// LS Electric XG5000 project: 0201 선풍기
// PLC LSPLC

PROGRAM NewProgram (task: 스캔 프로그램)

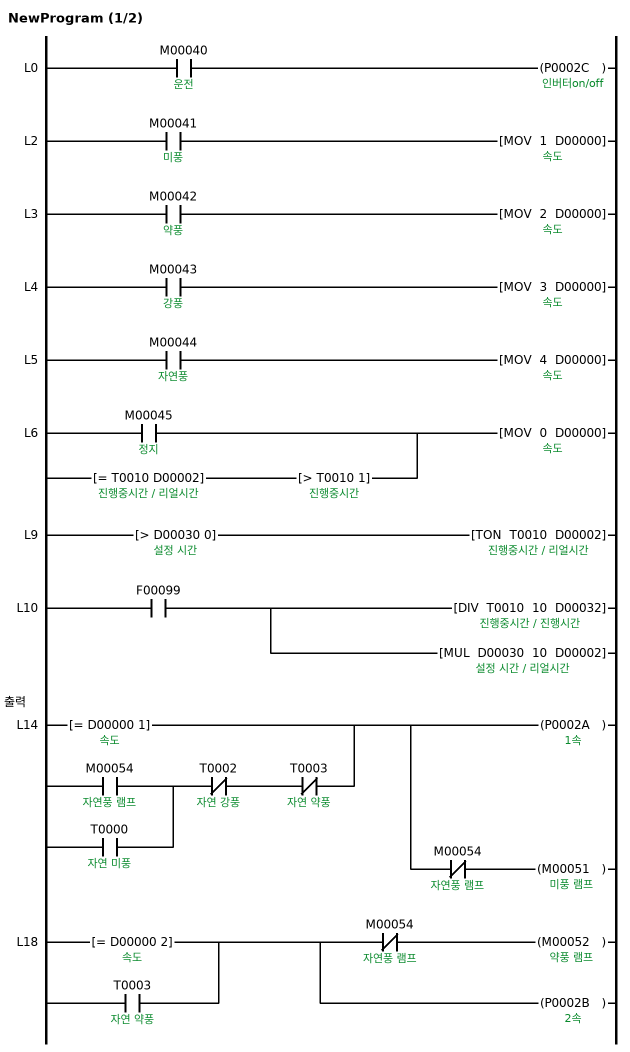
; L0
LOAD      M00040	// 운전
OUT       P0002C	// 인버터on/off
; L2
LOAD      M00041	// 미풍
MOV       1 D00000	// 속도
; L3
LOAD      M00042	// 약풍
MOV       2 D00000	// 속도
; L4
LOAD      M00043	// 강풍
MOV       3 D00000	// 속도
; L5
LOAD      M00044	// 자연풍
MOV       4 D00000	// 속도
; L6
LOAD      M00045	// 정지
LOAD=     T0010 D00002	// 진행중시간 / 리얼시간
AND>      T0010 1	// 진행중시간
OR LOAD
MOV       0 D00000	// 속도
; L9
LOAD>     D00030 0	// 설정 시간
TON       T0010 D00002	// 진행중시간 / 리얼시간
; L10
LOAD      F00099
DIV       T0010 10 D00032	// 진행중시간 / 진행시간
MUL       D00030 10 D00002	// 설정 시간 / 리얼시간
출력:
; L14
LOAD=     D00000 1	// 속도
LOAD      M00054	// 자연풍 램프
OR        T0000	// 자연 미풍
AND NOT   T0002	// 자연 강풍
AND NOT   T0003	// 자연 약풍
OR LOAD
OUT       P0002A	// 1속
AND NOT   M00054	// 자연풍 램프
OUT       M00051	// 미풍 램프
; L18
LOAD=     D00000 2	// 속도
OR        T0003	// 자연 약풍
MPUSH
AND NOT   M00054	// 자연풍 램프
OUT       M00052	// 약풍 램프
MPOP
OUT       P0002B	// 2속

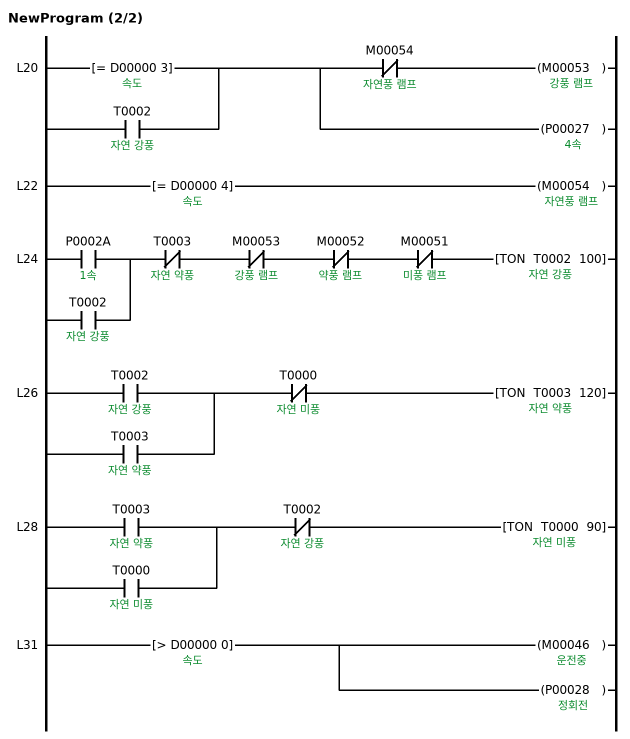
; L20
LOAD=     D00000 3	// 속도
OR        T0002	// 자연 강풍
MPUSH
AND NOT   M00054	// 자연풍 램프
OUT       M00053	// 강풍 램프
MPOP
OUT       P00027	// 4속
; L22
LOAD=     D00000 4	// 속도
OUT       M00054	// 자연풍 램프
; L24
LOAD      P0002A	// 1속
OR        T0002	// 자연 강풍
AND NOT   T0003	// 자연 약풍
AND NOT   M00053	// 강풍 램프
AND NOT   M00052	// 약풍 램프
AND NOT   M00051	// 미풍 램프
TON       T0002 100	// 자연 강풍
; L26
LOAD      T0002	// 자연 강풍
OR        T0003	// 자연 약풍
AND NOT   T0000	// 자연 미풍
TON       T0003 120	// 자연 약풍
; L28
LOAD      T0003	// 자연 약풍
OR        T0000	// 자연 미풍
AND NOT   T0002	// 자연 강풍
TON       T0000 90	// 자연 미풍
; L31
LOAD>     D00000 0	// 속도
OUT       M00046	// 운전중
OUT       P00028	// 정회전

VARIABLES AND COMMENTS (devices not used above)
M00001	BIT	정회전
M00002	BIT	역회전
P00006	BIT	출구
T0001	BIT/WORD	자연 미풍
D00100	WORD	표시 시간